{attribute 'GeneratedUsingTerminal: EK1122-0000-0018'}
{attribute addProperty BoxType "EK1122-0000-0018"}
{attribute addProperty Id "Beckhoff_ELXxxxxsub_EK1100EK1100_1FC0878B2"}
{attribute addProperty CRC "1071171527"}
{attribute addProperty Size "2"}
TYPE Beckhoff_ELXxxxxEK1122_3FD8C7C7 EXTENDS EK1122_1FC0878B :
STRUCT
	{attribute addProperty Name "Beckhoff_ELXxxxxsub_EK1100"}
	{attribute addProperty PreviousPort "Beckhoff ELXxxxxEK1122 : D"}
	Beckhoff_ELXxxxxsub_EK1100 : EK1100_1FC0878B;
END_STRUCT
END_TYPE

(* stored: Version 1.2.0.0, ProductVersion 3.1.4024.9
   DUT Beckhoff_ELXxxxxEK1122_3FD8C7C7: Id {f44d5e0a-6f2e-41e1-bee6-bc71ed1b4d0c} *)
